// TIA Portal project "voda" (V17)

(* hardware
DEVICE "S71500/ET200MP-Station_1"  S7-1500 station
   slot 0: "Profilschiene_0"  6ES7 590-1***0-0AA0
   slot 1: "PLC_1"  CPU 1511-1 PN  6ES7 511-1AK00-0AB0  V1.8
   slot 2: "AI 8xU/I/RTD/TC ST_1"  AI 8xU/I/RTD/TC ST  6ES7 531-7KF00-0AB0  V2.0
   slot 3: "AI 8xU/I/RTD/TC ST_2"  AI 8xU/I/RTD/TC ST  6ES7 531-7KF00-0AB0  V2.0
   slot 4: "AI 8xU/I/RTD/TC ST_3"  AI 8xU/I/RTD/TC ST  6ES7 531-7KF00-0AB0  V2.0
   slot 5: "AI 8xU/I/RTD/TC ST_4"  AI 8xU/I/RTD/TC ST  6ES7 531-7KF00-0AB0  V2.0
   slot 6: "DI 16x24VDC BA_1"  DI 16x24VDC BA  6ES7 521-1BH10-0AA0  V1.0
DEVICE "HMI_1"  KTP700 Basic PN
   slot 0: "HMI_1"  KTP700 Basic PN  6AV2 123-2GB03-0AX0  17.0.0.0
   slot 1: "HMI_RT_1"  KTP700 Basic PN  6AV2 123-2GB03-0AX0  17.0.0.0
   slot 5: "HMI_1.IE_CP_1"  PROFINET Interface  17.0.0.0
      slot 1: "PROFINET Interface_1"  PROFINET Interface
         slot 1: "Port_1"  Port
*)

// ===== PLC "PLC_1"  CPU 1511-1 PN =====

VAR_GLOBAL   // PLC tag table "Standard-Variablentabelle"
   "Start" AT %I0.0 : Bool;
   "Reset" AT %I0.1 : Bool;
   "Stop" AT %I0.2 : Bool;
   "Factory_I/O" AT %I0.3 : Bool;
   "Level_Meter" AT %ID30 : Real;
   "Flow_Meter" AT %ID34 : Real;
   "Set_Point" AT %ID38 : Real;
   "Start_Light" AT %Q0.0 : Bool;
   "Reset_Light" AT %Q0.1 : Bool;
   "Stop_Light" AT %Q0.2 : Bool;
   "Fill_valve" AT %QD30 : Real;
   "Discharge_valve" AT %QD34 : Real;
   "SP" AT %QD38 : DInt;
   "PV" AT %QD42 : DInt;
   "Tag_1" AT %M0.0 : Bool;
   "Tag_2" AT %M100.2 : Bool;
   "Tag_3" AT %M600.0 : Bool;
   "Tag_4" AT %M20.0 : Bool;
   "Tag_5" AT %M20.1 : Bool;
   "Tag_6" AT %M20.2 : Bool;
END_VAR

DATA_BLOCK "global"   // DB1
{ S7_Optimized_Access := 'TRUE' }
VERSION : 0.1
   VAR
      POM : Array[0..100] of Bool;
      POM_BR : Array[0..100] of Real;
      SP_Real : Real;
      PV_Real : Real;
      Kp_Level : Real;
      Ki_Level : Real;
      Kp_Flow : Real;
      Ki_Flow : Real;
      Flow_Real : Real;
      Discharge_Real : Real;
      SP_flow : Real;
      "LevelSetPoint%" : Real;
      "FlowSP%" : Real;
      "FlowPV%" : Real;
      "LevelPV%" : Real;
      PV_flow : Real;
      FactoryIOPTrig : Bool;
      PID_CompactMode : Int := 3;
      "FlowSP0-10" : Real;
   END_VAR
BEGIN
END_DATA_BLOCK

DATA_BLOCK "PID_Level"   // DB2
{ S7_Optimized_Access := 'TRUE' }
VERSION : 0.1
// stored: InstanceOfName Block_3
"Block_3"
BEGIN
END_DATA_BLOCK

DATA_BLOCK "PID_Flow"   // DB3
{ S7_Optimized_Access := 'TRUE' }
VERSION : 0.1
// stored: InstanceOfName Block_3
"Block_3"
BEGIN
END_DATA_BLOCK

DATA_BLOCK "HMI Tags"   // DB7
{ S7_Optimized_Access := 'TRUE' }
VERSION : 0.1
   VAR
      PV_Level : Real;
      SP_Level : Real;
      "SP_Flow%" : DInt;
      PV_Flow : DInt;
      "SP_Level%" : Real;
      LevelSetPointInCM : Bool;
      "LevelSetPointIn%" : Bool;
      LevelSetpointInCMButton : Bool;
      "LevelSetpointIn%Button" : Bool;
      HMIButton : Bool;
      FactoryIOButton : Bool;
      HMI : Bool;
      FactoryIO : Bool;
      HMISPLevelSet : Real;
      "HMISPLevelSet%" : Real;
      "Dozvoljeno%" : Bool;
      DozvoljenoCM : Bool;
      Warning : Bool;
      LL_Alarm : Bool;
      L_Alarm : Bool;
      H_Alarm : Bool;
      HH_Alarm : Bool;
      LL_Pom : Bool;
      Level_0 : Bool;
      HH_Pom : Bool;
      ACKButton : Bool;
      ACK : Bool;
   END_VAR
BEGIN
END_DATA_BLOCK

FUNCTION_BLOCK "Block_3"   // FB1, SCL
{ S7_Optimized_Access := 'TRUE' }
VERSION : 0.1
   VAR_INPUT
      SP : Real;
      PV : Real;
      Kp : Real;
      Ki : Real;
      Xi_max : Real;
      "dt" : Real;
      Xi_min : Real;
   END_VAR
   VAR_OUTPUT
      U : Real;
   END_VAR
   VAR
      I : Real;
      Xi : Real;
      error : Real;
   END_VAR
BEGIN
   #I := 0;
   #error := #SP - #PV;
   #I := #I + #error * #dt;
   #Xi := (#Kp * #error) + (#Ki * #I);
   IF #Xi > #Xi_max THEN
       #U := #Xi_max;
       #I := #I - #error * #dt;
   ELSIF #Xi < #Xi_min THEN
       #U := #Xi_min;
       #I := #I - #error * #dt;
   ELSE
       #U := #Xi;
   END_IF;
END_FUNCTION_BLOCK

FUNCTION "Block_1" : Void   // FC1, LAD
{ S7_Optimized_Access := 'TRUE' }
VERSION : 0.1
   VAR_TEMP   // added for the SCL form of the ladder/FBD networks
      _w1 : Bool;
      _w2 : Bool;
   END_VAR
BEGIN

REGION Network 1
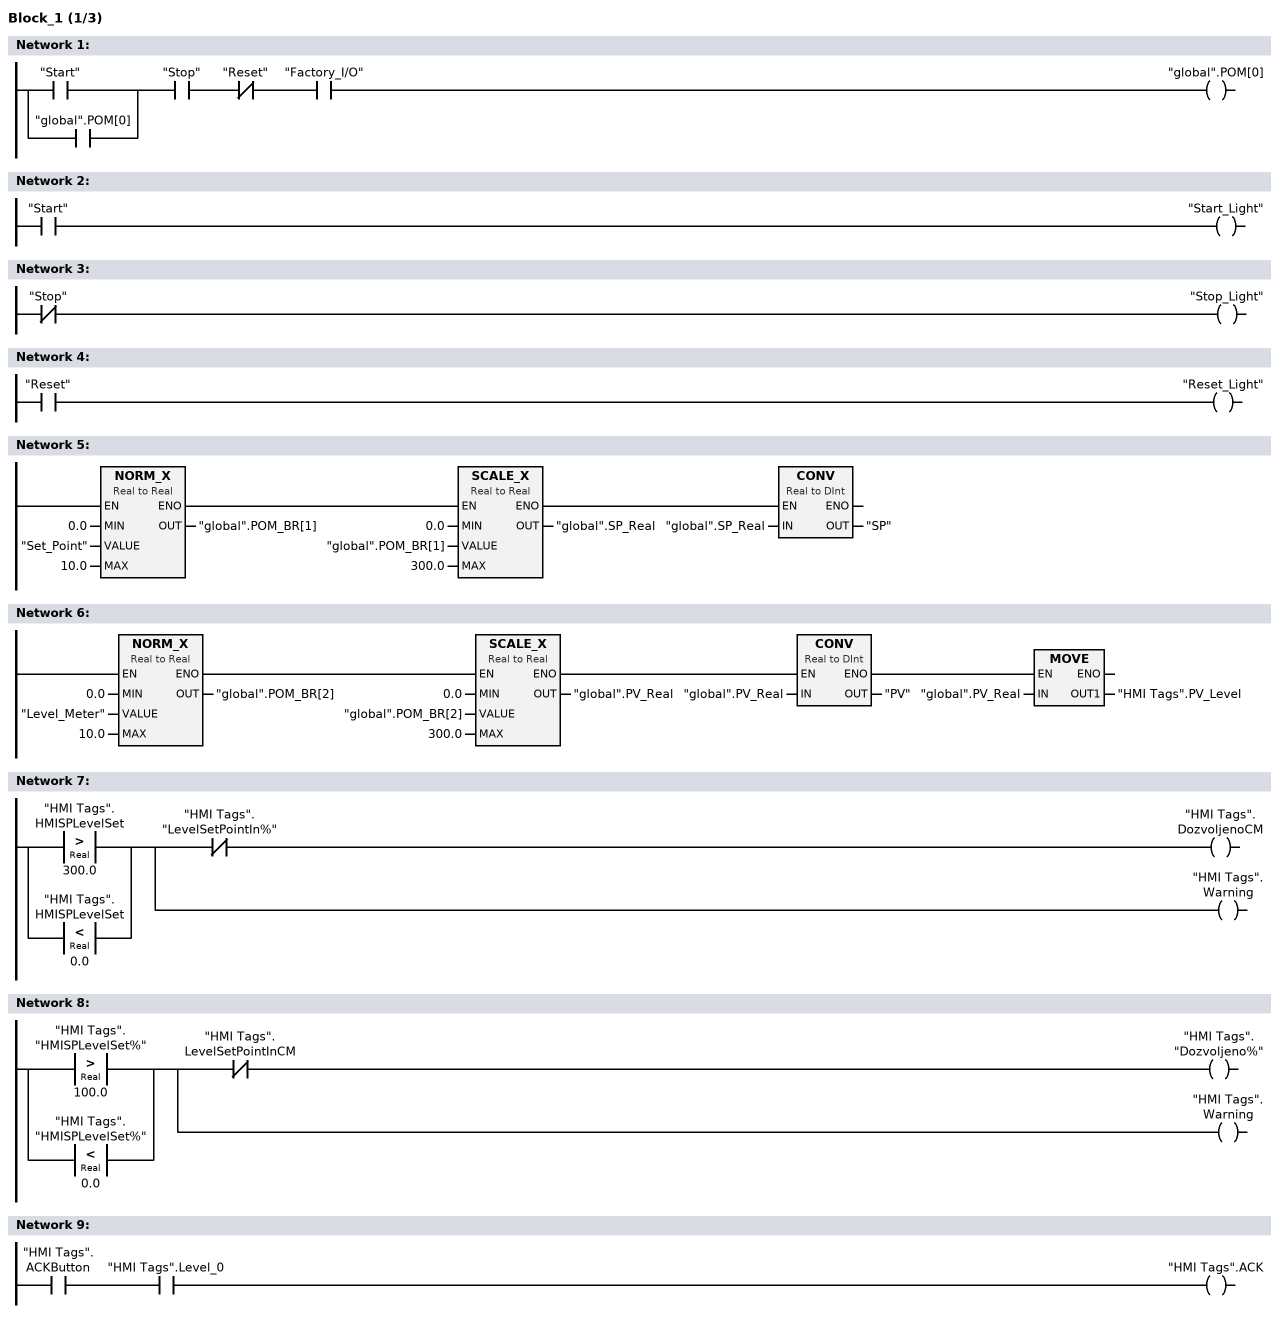
   RUNG wire#powerrail
      Contact( "Start" )
      wire#w1
      Contact( "Stop" )
      I_Contact( "Reset" )
      Contact( "Factory_I/O" )
      Coil( "global".POM[0] )
   END_RUNG
   RUNG wire#powerrail
      Contact( "global".POM[0] )
   END_RUNG wire#w1
   // the same network as SCL:
   "global".POM[0] := ("Start" OR "global".POM[0]) AND "Stop" AND NOT "Reset" AND "Factory_I/O";
END_REGION

REGION Network 2
   RUNG wire#powerrail
      Contact( "Start" )
      Coil( "Start_Light" )
   END_RUNG
   // the same network as SCL:
   "Start_Light" := "Start";
END_REGION

REGION Network 3
   RUNG wire#powerrail
      I_Contact( "Stop" )
      Coil( "Stop_Light" )
   END_RUNG
   // the same network as SCL:
   "Stop_Light" := NOT "Stop";
END_REGION

REGION Network 4
   RUNG wire#powerrail
      Contact( "Reset" )
      Coil( "Reset_Light" )
   END_RUNG
   // the same network as SCL:
   "Reset_Light" := "Reset";
END_REGION

REGION Network 5
   RUNG wire#powerrail
      { S7_Templates := "[SrcType := Real, DestType := Real]" } Normalize(min := 0.0, value := "Set_Point", max := 10.0, out => "global".POM_BR[1])
      { S7_Templates := "[SrcType := Real, DestType := Real]" } Scale(min := 0.0, value := "global".POM_BR[1], max := 300.0, out => "global".SP_Real)
      { S7_Templates := "[SrcType := Real, DestType := DInt]" } Convert(in := "global".SP_Real, out => "SP")
   END_RUNG
   // the same network as SCL:
   "global".POM_BR[1] := NORM_X(MIN := 0.0, VALUE := "Set_Point", MAX := 10.0);
   "global".SP_Real := SCALE_X(MIN := 0.0, VALUE := "global".POM_BR[1], MAX := 300.0);
   "SP" := REAL_TO_DINT("global".SP_Real);
END_REGION

REGION Network 6
   RUNG wire#powerrail
      { S7_Templates := "[SrcType := Real, DestType := Real]" } Normalize(min := 0.0, value := "Level_Meter", max := 10.0, out => "global".POM_BR[2])
      { S7_Templates := "[SrcType := Real, DestType := Real]" } Scale(min := 0.0, value := "global".POM_BR[2], max := 300.0, out => "global".PV_Real)
      { S7_Templates := "[SrcType := Real, DestType := DInt]" } Convert(in := "global".PV_Real, out => "PV")
      Move(in := "global".PV_Real, out1 => "HMI Tags".PV_Level)
   END_RUNG
   // the same network as SCL:
   "global".POM_BR[2] := NORM_X(MIN := 0.0, VALUE := "Level_Meter", MAX := 10.0);
   "global".PV_Real := SCALE_X(MIN := 0.0, VALUE := "global".POM_BR[2], MAX := 300.0);
   "PV" := REAL_TO_DINT("global".PV_Real);
   "HMI Tags".PV_Level := "global".PV_Real;
END_REGION

REGION Network 7
   RUNG wire#powerrail
      { S7_Templates := "SrcType := Real" } GT_Contact(in1 := "HMI Tags".HMISPLevelSet, in2 := 300.0)
      wire#w1
      I_Contact( "HMI Tags"."LevelSetPointIn%" )
      Coil( "HMI Tags".DozvoljenoCM )
   END_RUNG
   RUNG wire#powerrail
      { S7_Templates := "SrcType := Real" } LT_Contact(in1 := "HMI Tags".HMISPLevelSet, in2 := 0.0)
   END_RUNG wire#w1
   RUNG wire#w1
      Coil( "HMI Tags".Warning )
   END_RUNG
   // the same network as SCL:
   #_w1 := ("HMI Tags".HMISPLevelSet > 300.0) OR ("HMI Tags".HMISPLevelSet < 0.0);
   "HMI Tags".DozvoljenoCM := #_w1 AND NOT "HMI Tags"."LevelSetPointIn%";
   "HMI Tags".Warning := #_w1;
END_REGION

REGION Network 8
   RUNG wire#powerrail
      { S7_Templates := "SrcType := Real" } GT_Contact(in1 := "HMI Tags"."HMISPLevelSet%", in2 := 100.0)
      wire#w1
      I_Contact( "HMI Tags".LevelSetPointInCM )
      Coil( "HMI Tags"."Dozvoljeno%" )
   END_RUNG
   RUNG wire#powerrail
      { S7_Templates := "SrcType := Real" } LT_Contact(in1 := "HMI Tags"."HMISPLevelSet%", in2 := 0.0)
   END_RUNG wire#w1
   RUNG wire#w1
      Coil( "HMI Tags".Warning )
   END_RUNG
   // the same network as SCL:
   #_w1 := ("HMI Tags"."HMISPLevelSet%" > 100.0) OR ("HMI Tags"."HMISPLevelSet%" < 0.0);
   "HMI Tags"."Dozvoljeno%" := #_w1 AND NOT "HMI Tags".LevelSetPointInCM;
   "HMI Tags".Warning := #_w1;
END_REGION

REGION Network 9
   RUNG wire#powerrail
      Contact( "HMI Tags".ACKButton )
      Contact( "HMI Tags".Level_0 )
      Coil( "HMI Tags".ACK )
   END_RUNG
   // the same network as SCL:
   "HMI Tags".ACK := "HMI Tags".ACKButton AND "HMI Tags".Level_0;
END_REGION

REGION Network 10
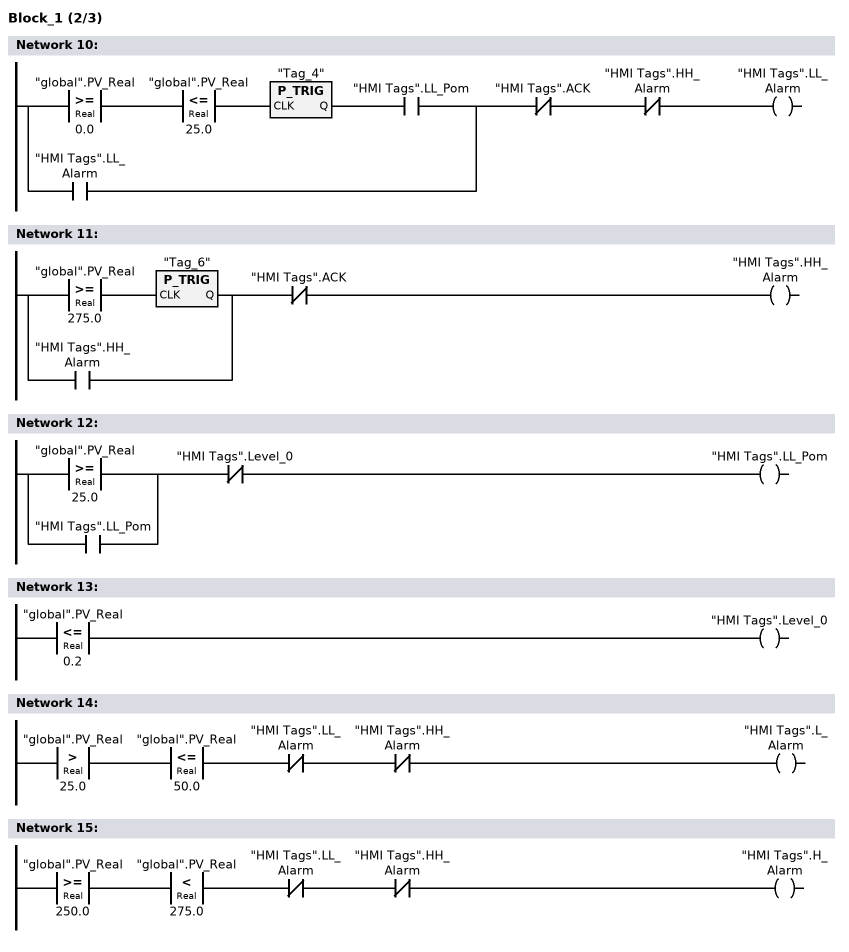
   RUNG wire#powerrail
      { S7_Templates := "SrcType := Real" } GE_Contact(in1 := "global".PV_Real, in2 := 0.0)
      { S7_Templates := "SrcType := Real" } LE_Contact(in1 := "global".PV_Real, in2 := 25.0)
      P_Trig( "Tag_4" )
      Contact( "HMI Tags".LL_Pom )
      wire#w1
      I_Contact( "HMI Tags".ACK )
      I_Contact( "HMI Tags".HH_Alarm )
      Coil( "HMI Tags".LL_Alarm )
   END_RUNG
   RUNG wire#powerrail
      Contact( "HMI Tags".LL_Alarm )
   END_RUNG wire#w1
   // the same network as SCL:
   #_w1 := ("global".PV_Real >= 0.0) AND ("global".PV_Real <= 25.0);
   #_w2 := #_w1 AND NOT "Tag_4";   // rising edge
   "Tag_4" := #_w1;
   "HMI Tags".LL_Alarm := ((#_w2 AND "HMI Tags".LL_Pom) OR "HMI Tags".LL_Alarm) AND NOT "HMI Tags".ACK AND NOT "HMI Tags".HH_Alarm;
END_REGION

REGION Network 11
   RUNG wire#powerrail
      { S7_Templates := "SrcType := Real" } GE_Contact(in1 := "global".PV_Real, in2 := 275.0)
      P_Trig( "Tag_6" )
      wire#w1
      I_Contact( "HMI Tags".ACK )
      Coil( "HMI Tags".HH_Alarm )
   END_RUNG
   RUNG wire#powerrail
      Contact( "HMI Tags".HH_Alarm )
   END_RUNG wire#w1
   // the same network as SCL:
   #_w1 := "global".PV_Real >= 275.0;
   #_w2 := #_w1 AND NOT "Tag_6";   // rising edge
   "Tag_6" := #_w1;
   "HMI Tags".HH_Alarm := (#_w2 OR "HMI Tags".HH_Alarm) AND NOT "HMI Tags".ACK;
END_REGION

REGION Network 12
   RUNG wire#powerrail
      { S7_Templates := "SrcType := Real" } GE_Contact(in1 := "global".PV_Real, in2 := 25.0)
      wire#w1
      I_Contact( "HMI Tags".Level_0 )
      Coil( "HMI Tags".LL_Pom )
   END_RUNG
   RUNG wire#powerrail
      Contact( "HMI Tags".LL_Pom )
   END_RUNG wire#w1
   // the same network as SCL:
   "HMI Tags".LL_Pom := (("global".PV_Real >= 25.0) OR "HMI Tags".LL_Pom) AND NOT "HMI Tags".Level_0;
END_REGION

REGION Network 13
   RUNG wire#powerrail
      { S7_Templates := "SrcType := Real" } LE_Contact(in1 := "global".PV_Real, in2 := 0.2)
      Coil( "HMI Tags".Level_0 )
   END_RUNG
   // the same network as SCL:
   "HMI Tags".Level_0 := "global".PV_Real <= 0.2;
END_REGION

REGION Network 14
   RUNG wire#powerrail
      { S7_Templates := "SrcType := Real" } GT_Contact(in1 := "global".PV_Real, in2 := 25.0)
      { S7_Templates := "SrcType := Real" } LE_Contact(in1 := "global".PV_Real, in2 := 50.0)
      I_Contact( "HMI Tags".LL_Alarm )
      I_Contact( "HMI Tags".HH_Alarm )
      Coil( "HMI Tags".L_Alarm )
   END_RUNG
   // the same network as SCL:
   "HMI Tags".L_Alarm := ("global".PV_Real > 25.0) AND ("global".PV_Real <= 50.0) AND NOT "HMI Tags".LL_Alarm AND NOT "HMI Tags".HH_Alarm;
END_REGION

REGION Network 15
   RUNG wire#powerrail
      { S7_Templates := "SrcType := Real" } GE_Contact(in1 := "global".PV_Real, in2 := 250.0)
      { S7_Templates := "SrcType := Real" } LT_Contact(in1 := "global".PV_Real, in2 := 275.0)
      I_Contact( "HMI Tags".LL_Alarm )
      I_Contact( "HMI Tags".HH_Alarm )
      Coil( "HMI Tags".H_Alarm )
   END_RUNG
   // the same network as SCL:
   "HMI Tags".H_Alarm := ("global".PV_Real >= 250.0) AND ("global".PV_Real < 275.0) AND NOT "HMI Tags".LL_Alarm AND NOT "HMI Tags".HH_Alarm;
END_REGION

REGION Network 16
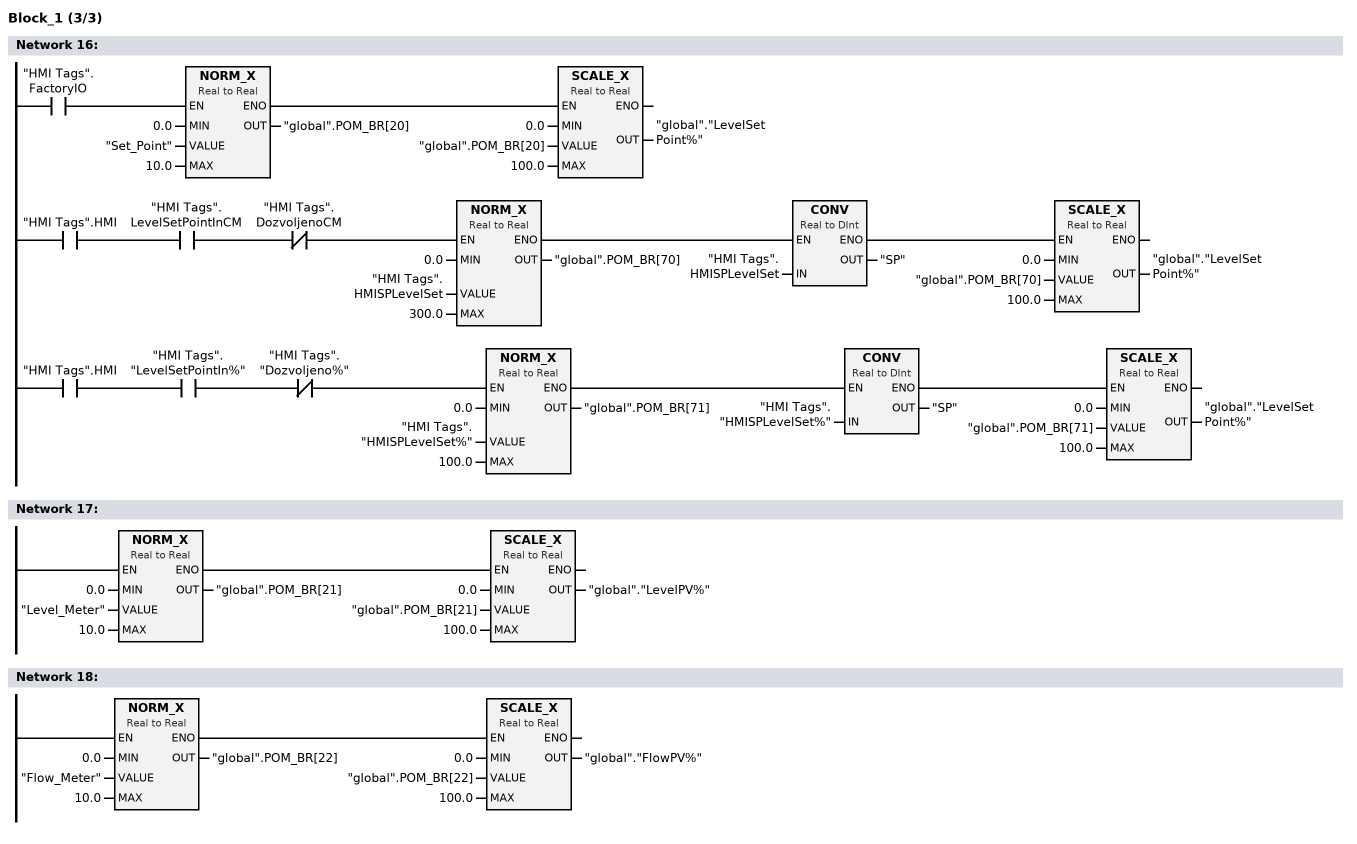
   RUNG wire#powerrail
      Contact( "HMI Tags".FactoryIO )
      { S7_Templates := "[SrcType := Real, DestType := Real]" } Normalize(min := 0.0, value := "Set_Point", max := 10.0, out => "global".POM_BR[20])
      { S7_Templates := "[SrcType := Real, DestType := Real]" } Scale(min := 0.0, value := "global".POM_BR[20], max := 100.0, out => "global"."LevelSetPoint%")
   END_RUNG
   RUNG wire#powerrail
      Contact( "HMI Tags".HMI )
      Contact( "HMI Tags".LevelSetPointInCM )
      I_Contact( "HMI Tags".DozvoljenoCM )
      { S7_Templates := "[SrcType := Real, DestType := Real]" } Normalize(min := 0.0, value := "HMI Tags".HMISPLevelSet, max := 300.0, out => "global".POM_BR[70])
      { S7_Templates := "[SrcType := Real, DestType := DInt]" } Convert(in := "HMI Tags".HMISPLevelSet, out => "SP")
      { S7_Templates := "[SrcType := Real, DestType := Real]" } Scale(min := 0.0, value := "global".POM_BR[70], max := 100.0, out => "global"."LevelSetPoint%")
   END_RUNG
   RUNG wire#powerrail
      Contact( "HMI Tags".HMI )
      Contact( "HMI Tags"."LevelSetPointIn%" )
      I_Contact( "HMI Tags"."Dozvoljeno%" )
      { S7_Templates := "[SrcType := Real, DestType := Real]" } Normalize(min := 0.0, value := "HMI Tags"."HMISPLevelSet%", max := 100.0, out => "global".POM_BR[71])
      { S7_Templates := "[SrcType := Real, DestType := DInt]" } Convert(in := "HMI Tags"."HMISPLevelSet%", out => "SP")
      { S7_Templates := "[SrcType := Real, DestType := Real]" } Scale(min := 0.0, value := "global".POM_BR[71], max := 100.0, out => "global"."LevelSetPoint%")
   END_RUNG
   // the same network as SCL:
   IF "HMI Tags".FactoryIO THEN
       "global".POM_BR[20] := NORM_X(MIN := 0.0, VALUE := "Set_Point", MAX := 10.0);
       "global"."LevelSetPoint%" := SCALE_X(MIN := 0.0, VALUE := "global".POM_BR[20], MAX := 100.0);
   END_IF;
   IF "HMI Tags".HMI AND "HMI Tags".LevelSetPointInCM AND NOT "HMI Tags".DozvoljenoCM THEN
       "global".POM_BR[70] := NORM_X(MIN := 0.0, VALUE := "HMI Tags".HMISPLevelSet, MAX := 300.0);
       "SP" := REAL_TO_DINT("HMI Tags".HMISPLevelSet);
       "global"."LevelSetPoint%" := SCALE_X(MIN := 0.0, VALUE := "global".POM_BR[70], MAX := 100.0);
   END_IF;
   IF "HMI Tags".HMI AND "HMI Tags"."LevelSetPointIn%" AND NOT "HMI Tags"."Dozvoljeno%" THEN
       "global".POM_BR[71] := NORM_X(MIN := 0.0, VALUE := "HMI Tags"."HMISPLevelSet%", MAX := 100.0);
       "SP" := REAL_TO_DINT("HMI Tags"."HMISPLevelSet%");
       "global"."LevelSetPoint%" := SCALE_X(MIN := 0.0, VALUE := "global".POM_BR[71], MAX := 100.0);
   END_IF;
END_REGION

REGION Network 17
   RUNG wire#powerrail
      { S7_Templates := "[SrcType := Real, DestType := Real]" } Normalize(min := 0.0, value := "Level_Meter", max := 10.0, out => "global".POM_BR[21])
      { S7_Templates := "[SrcType := Real, DestType := Real]" } Scale(min := 0.0, value := "global".POM_BR[21], max := 100.0, out => "global"."LevelPV%")
   END_RUNG
   // the same network as SCL:
   "global".POM_BR[21] := NORM_X(MIN := 0.0, VALUE := "Level_Meter", MAX := 10.0);
   "global"."LevelPV%" := SCALE_X(MIN := 0.0, VALUE := "global".POM_BR[21], MAX := 100.0);
END_REGION

REGION Network 18
   RUNG wire#powerrail
      { S7_Templates := "[SrcType := Real, DestType := Real]" } Normalize(min := 0.0, value := "Flow_Meter", max := 10.0, out => "global".POM_BR[22])
      { S7_Templates := "[SrcType := Real, DestType := Real]" } Scale(min := 0.0, value := "global".POM_BR[22], max := 100.0, out => "global"."FlowPV%")
   END_RUNG
   // the same network as SCL:
   "global".POM_BR[22] := NORM_X(MIN := 0.0, VALUE := "Flow_Meter", MAX := 10.0);
   "global"."FlowPV%" := SCALE_X(MIN := 0.0, VALUE := "global".POM_BR[22], MAX := 100.0);
END_REGION
END_FUNCTION

FUNCTION "HMI" : Void   // FC2, LAD
{ S7_Optimized_Access := 'TRUE' }
VERSION : 0.1
BEGIN

REGION Network 1
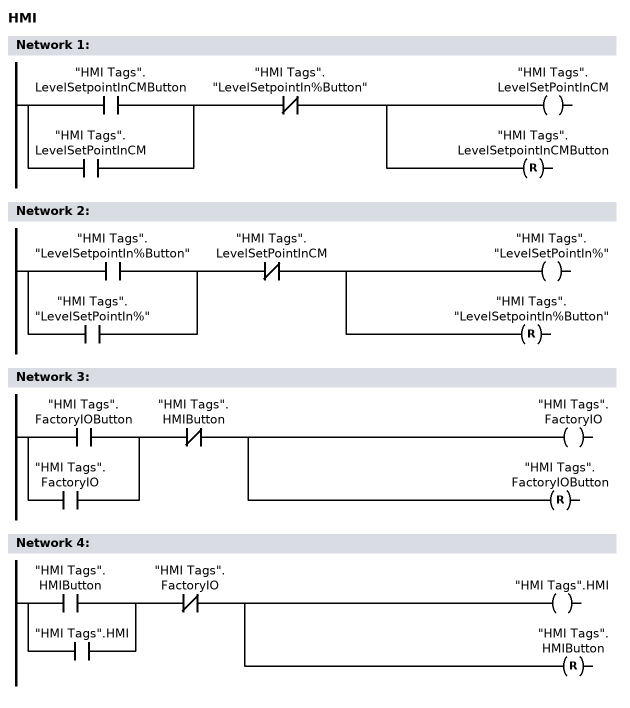
   RUNG wire#powerrail
      Contact( "HMI Tags".LevelSetpointInCMButton )
      wire#w1
      I_Contact( "HMI Tags"."LevelSetpointIn%Button" )
      wire#w2
      Coil( "HMI Tags".LevelSetPointInCM )
   END_RUNG
   RUNG wire#powerrail
      Contact( "HMI Tags".LevelSetPointInCM )
   END_RUNG wire#w1
   RUNG wire#w2
      R_Coil( "HMI Tags".LevelSetpointInCMButton )
   END_RUNG
   // the same network as SCL:
   "HMI Tags".LevelSetPointInCM := ("HMI Tags".LevelSetpointInCMButton OR "HMI Tags".LevelSetPointInCM) AND NOT "HMI Tags"."LevelSetpointIn%Button";
   IF "HMI Tags".LevelSetPointInCM THEN "HMI Tags".LevelSetpointInCMButton := FALSE; END_IF;
END_REGION

REGION Network 2
   RUNG wire#powerrail
      Contact( "HMI Tags"."LevelSetpointIn%Button" )
      wire#w1
      I_Contact( "HMI Tags".LevelSetPointInCM )
      wire#w2
      Coil( "HMI Tags"."LevelSetPointIn%" )
   END_RUNG
   RUNG wire#powerrail
      Contact( "HMI Tags"."LevelSetPointIn%" )
   END_RUNG wire#w1
   RUNG wire#w2
      R_Coil( "HMI Tags"."LevelSetpointIn%Button" )
   END_RUNG
   // the same network as SCL:
   "HMI Tags"."LevelSetPointIn%" := ("HMI Tags"."LevelSetpointIn%Button" OR "HMI Tags"."LevelSetPointIn%") AND NOT "HMI Tags".LevelSetPointInCM;
   IF "HMI Tags"."LevelSetPointIn%" THEN "HMI Tags"."LevelSetpointIn%Button" := FALSE; END_IF;
END_REGION

REGION Network 3
   RUNG wire#powerrail
      Contact( "HMI Tags".FactoryIOButton )
      wire#w1
      I_Contact( "HMI Tags".HMIButton )
      wire#w2
      Coil( "HMI Tags".FactoryIO )
   END_RUNG
   RUNG wire#powerrail
      Contact( "HMI Tags".FactoryIO )
   END_RUNG wire#w1
   RUNG wire#w2
      R_Coil( "HMI Tags".FactoryIOButton )
   END_RUNG
   // the same network as SCL:
   "HMI Tags".FactoryIO := ("HMI Tags".FactoryIOButton OR "HMI Tags".FactoryIO) AND NOT "HMI Tags".HMIButton;
   IF "HMI Tags".FactoryIO THEN "HMI Tags".FactoryIOButton := FALSE; END_IF;
END_REGION

REGION Network 4
   RUNG wire#powerrail
      Contact( "HMI Tags".HMIButton )
      wire#w1
      I_Contact( "HMI Tags".FactoryIO )
      wire#w2
      Coil( "HMI Tags".HMI )
   END_RUNG
   RUNG wire#powerrail
      Contact( "HMI Tags".HMI )
   END_RUNG wire#w1
   RUNG wire#w2
      R_Coil( "HMI Tags".HMIButton )
   END_RUNG
   // the same network as SCL:
   "HMI Tags".HMI := ("HMI Tags".HMIButton OR "HMI Tags".HMI) AND NOT "HMI Tags".FactoryIO;
   IF "HMI Tags".HMI THEN "HMI Tags".HMIButton := FALSE; END_IF;
END_REGION
END_FUNCTION

FUNCTION "MHJ-PLC-Lab-Function-S71500" : Void   // FC9000, SCL
{ S7_Optimized_Access := 'TRUE' }
VERSION : 0.1
   VAR_TEMP
      Value : Byte;
      ForCounter : Int;
   END_VAR
   VAR CONSTANT
      Value_01_DW : DWord := 16#1223_5486;
      Value_02_DW : DWord := 16#A6C9_D1F5;
   END_VAR
BEGIN

   #Value:=PEEK(area := 16#82,
        dbNumber := 0,
        byteOffset := 511);
   #Value := #Value + 1;

   POKE(area := 16#82,
        dbNumber := 0,
        byteOffset := 511,
        value := #Value);

   POKE(area := 16#82,
        dbNumber := 0,
        byteOffset := 1016,
        value := #Value_01_DW);
   POKE(area := 16#82,
        dbNumber := 0,
        byteOffset := 1020,
        value := #Value_02_DW);

   FOR #ForCounter := 0 TO 63 DO
       #Value:=PEEK(area := 16#1,
            dbNumber := 0,
            byteOffset := #ForCounter);
       POKE(area := 16#81,
            dbNumber := 0,
            byteOffset := #ForCounter,
            value := #Value);
   END_FOR;
   #Value := PEEK(area := 16#1,
                  dbNumber := 0,
                  byteOffset := 512);
   POKE(area := 16#82,
        dbNumber := 0,
        byteOffset := 512,
        value := #Value);
END_FUNCTION

ORGANIZATION_BLOCK "Main"   // OB1, FBD, ProgramCycle
TITLE = "Main Program Sweep (Cycle)"
{ S7_Optimized_Access := 'TRUE' }
VERSION : 0.1
   VAR_INPUT
      Initial_Call : Bool;   // Initial call of this OB
      Remanence : Bool;   // =True, if remanent data are available
   END_VAR
BEGIN

REGION Network 1
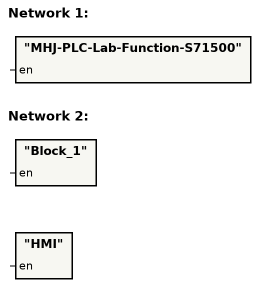
   "MHJ-PLC-Lab-Function-S71500"();
END_REGION

REGION Network 2
   "Block_1"();
   "HMI"();
END_REGION
END_ORGANIZATION_BLOCK

ORGANIZATION_BLOCK "PI kontroler"   // OB30, LAD, CyclicInterrupt
{ S7_Optimized_Access := 'TRUE' }
VERSION : 0.1
   VAR_INPUT
      Initial_Call : Bool;   // Initial call of this OB
      Event_Count : Int;   // Events discarded
   END_VAR
   VAR_TEMP   // added for the SCL form of the ladder/FBD networks
      _w1 : Bool;
   END_VAR
BEGIN

REGION Network 1
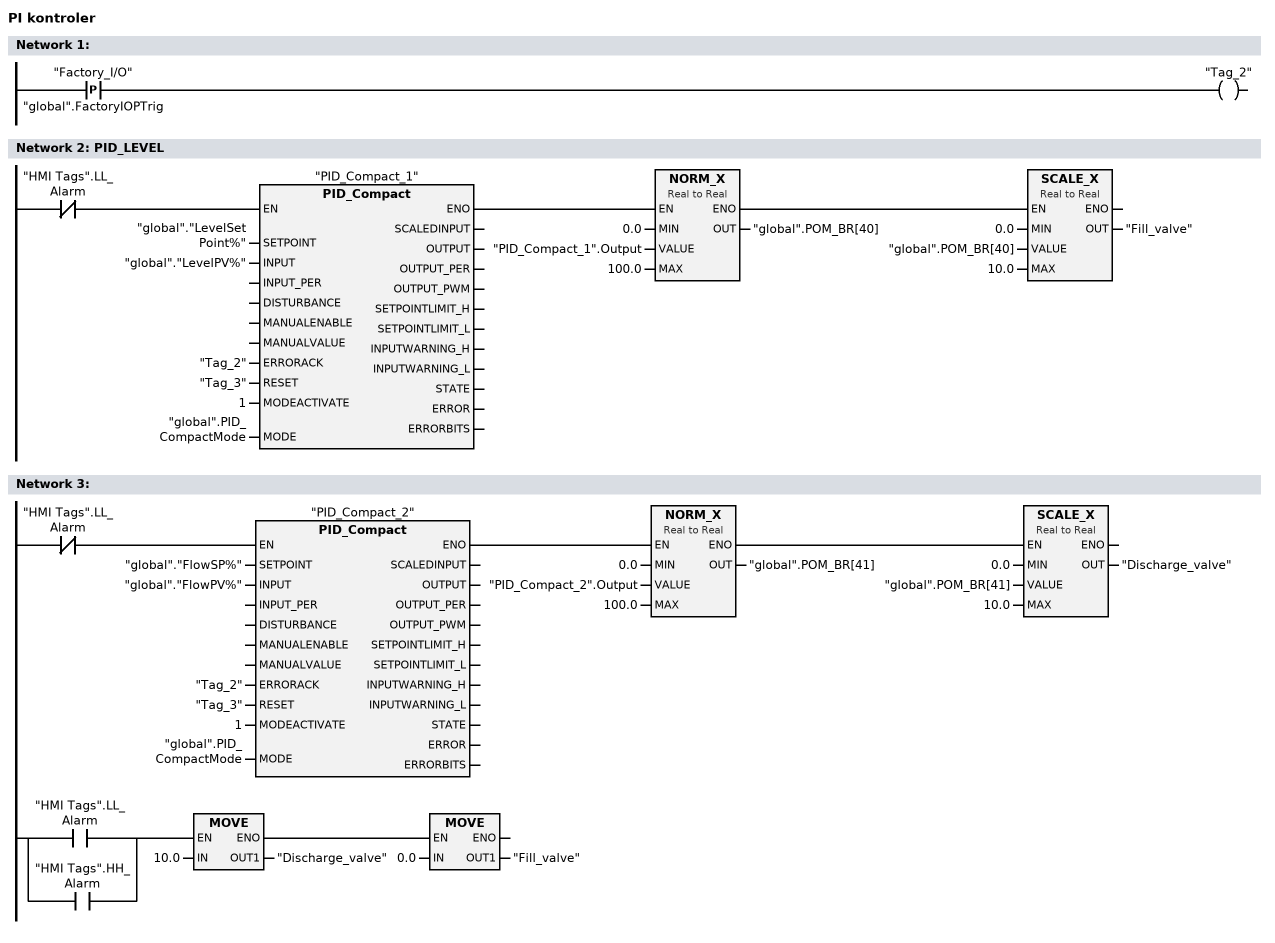
   RUNG wire#powerrail
      P_Contact(operand := "Factory_I/O", bit := "global".FactoryIOPTrig)
      Coil( "Tag_2" )
   END_RUNG
   // the same network as SCL:
   #_w1 := "Factory_I/O" AND NOT "global".FactoryIOPTrig;   // rising edge of "Factory_I/O"
   "global".FactoryIOPTrig := "Factory_I/O";
   "Tag_2" := #_w1;
END_REGION

REGION Network 2: PID_LEVEL
   // ENO of a box is taken as its EN; it also drops when the box reports an error
   #_w1 := NOT "HMI Tags".LL_Alarm;
   IF #_w1 THEN
       "PID_Compact_1"(Setpoint := "global"."LevelSetPoint%",   // PID_Compact
                       Input := "global"."LevelPV%",
                       ErrorAck := "Tag_2",
                       Reset := "Tag_3",
                       ModeActivate := 1,
                       Mode := "global".PID_CompactMode);
       "global".POM_BR[40] := NORM_X(MIN := 0.0, VALUE := "PID_Compact_1".Output, MAX := 100.0);
       "Fill_valve" := SCALE_X(MIN := 0.0, VALUE := "global".POM_BR[40], MAX := 10.0);
   END_IF;
END_REGION

REGION Network 3
   // ENO of a box is taken as its EN; it also drops when the box reports an error
   #_w1 := NOT "HMI Tags".LL_Alarm;
   IF #_w1 THEN
       "PID_Compact_2"(Setpoint := "global"."FlowSP%",   // PID_Compact
                       Input := "global"."FlowPV%",
                       ErrorAck := "Tag_2",
                       Reset := "Tag_3",
                       ModeActivate := 1,
                       Mode := "global".PID_CompactMode);
       "global".POM_BR[41] := NORM_X(MIN := 0.0, VALUE := "PID_Compact_2".Output, MAX := 100.0);
       "Discharge_valve" := SCALE_X(MIN := 0.0, VALUE := "global".POM_BR[41], MAX := 10.0);
   END_IF;
   IF "HMI Tags".LL_Alarm OR "HMI Tags".HH_Alarm THEN
       "Discharge_valve" := 10.0;
       "Fill_valve" := 0.0;
   END_IF;
END_REGION
END_ORGANIZATION_BLOCK

(* ===== HMI "HMI_RT_1" =====
system functions are stored by id; their names below are inferred from use
connection "Connection_1": ETHERNET, SMART_S7_1200_OMS
connection "HMI_Connection_1": ETHERNET, SMART_S7_1500_OMS

HMI tags "Default tag table"
   "HMI Tags_PV_Level" : Real = PLC "HMI Tags".PV_Level, 1 s
   "HMI Tags_SP_Level" : Real = PLC "HMI Tags".SP_Level, 1 s
   "HMI Tags_SP_Level%" : Real = PLC "HMI Tags".SP_Level%, 1 s
   "HMI Tags_LevelSetpointInCMButton" : Bool = PLC "HMI Tags".LevelSetpointInCMButton, 1 s
   "HMI Tags_HMI/FIO" : Bool = PLC "HMI Tags".HMIButton, 1 s
   "HMI Tags_FactoryIOButton" : Bool = PLC "HMI Tags".FactoryIOButton, 1 s
   "HMI Tags_HMISPLevelSet" : Real = PLC "HMI Tags".HMISPLevelSet, 1 s
   "HMI Tags_LevelSetpointIn%Button" : Bool = PLC "HMI Tags".LevelSetpointIn%Button, 1 s
   "HMI Tags_LevelSetPointInCM" : Bool = PLC "HMI Tags".LevelSetPointInCM, 1 s
   "HMI Tags_LevelSetPointIn%" : Bool = PLC "HMI Tags".LevelSetPointIn%, 1 s
   "HMI Tags_HMISPLevelSet%" : Real = PLC "HMI Tags".HMISPLevelSet%, 1 s
   "HMI Tags_Dozvoljeno%" : Bool = PLC "HMI Tags".Dozvoljeno%, 1 s
   "HMI Tags_DozvoljenoCM" : Bool = PLC "HMI Tags".DozvoljenoCM, 1 s
   "HMI Tags_FactoryIO" : Bool = PLC "HMI Tags".FactoryIO, 1 s
   "HMI Tags_HMI" : Bool = PLC "HMI Tags".HMI, 1 s
   "global_FlowSP%" : Real = PLC global.FlowSP%, 1 s
   "HMI Tags_Warning" : Bool = PLC "HMI Tags".Warning, 1 s
   "HMI Tags_LL_Alarm" : Bool = PLC "HMI Tags".LL_Alarm, 1 s
   "HMI Tags_L_Alarm" : Bool = PLC "HMI Tags".L_Alarm, 1 s
   "HMI Tags_H_Alarm" : Bool = PLC "HMI Tags".H_Alarm, 1 s
   "HMI Tags_HH_Alarm" : Bool = PLC "HMI Tags".HH_Alarm, 1 s
   "HMI Tags_ACK" : Bool = PLC "HMI Tags".ACK, 1 s
   "HMI Tags_ACKButton" : Bool = PLC "HMI Tags".ACKButton, 1 s
   "global_FlowPV%" : Real = PLC global.FlowPV%, 1 s
   "HMI Tags_LL_Pom" : Bool = PLC "HMI Tags".LL_Pom, 1 s

screen "Screen_1" 800x480
   GraphicView "Graphic view_1" at 44,86 size 267x322; Picture "Graphic_2"
   Bar "Bar_1" at 55,108 size 239x284; MinimumValue 0; MaximumValue 300
      ProcessValue <- "HMI Tags_PV_Level"
   IOField "I/O field_1" at 446,165 size 54x38; FormatPattern 999
      ProcessValue <- "HMI Tags_HMISPLevelSet"
      Visibility <- "HMI Tags_LevelSetPointInCM"
   TextField "Text field_1" at 431,134 size 102x20; Text 'Set Point in CM'
      Visibility <- "HMI Tags_LevelSetPointInCM"
   IOField "I/O field_2" at 337,165 size 66x39; FormatPattern 999
      ProcessValue <- "HMI Tags_PV_Level"
   TextField "Text field_2" at 328,134 size 95x20; Text 'Process value'
   Button "Button_1" at 364,365 size 136x62; TextOff 'HMI'
      on Click: SetBit("HMI Tags_HMI/FIO")
      Appearance <- "HMI Tags_HMI"
   Button "Button_2" at 364,270 size 136x62; TextOff 'Factory'
      on Click: SetBit("HMI Tags_FactoryIOButton")
      Appearance <- "HMI Tags_FactoryIO"
   Button "Button_3" at 611,365 size 136x62; TextOff 'IN CM'
      on Click: SetBit("HMI Tags_LevelSetpointInCMButton")
      Appearance <- "HMI Tags_LevelSetPointInCM"
   Button "Button_4" at 610,271 size 136x62; TextOff 'IN %'
      on Click: SetBit("HMI Tags_LevelSetpointIn%Button")
      Appearance <- "HMI Tags_LevelSetPointIn%"
   IOField "I/O field_3" at 446,165 size 60x38; FormatPattern 999
      ProcessValue <- "HMI Tags_HMISPLevelSet%"
      Visibility <- "HMI Tags_LevelSetPointIn%"
   TextField "Text field_3" at 431,134 size 97x20; Text 'Set Point in %'
      Visibility <- "HMI Tags_LevelSetPointIn%"
   IOField "I/O field_4" at 550,166 size 49x38; FormatPattern 999
      ProcessValue <- "global_FlowSP%"
   TextField "Text field_6" at 550,134 size 86x20; Text 'Flow SP in %'
   TextField "Text field_4" at 151,42 size 448x37; Text 'CHOOSE VALUE BETWEEN 0-100'
      Visibility <- "HMI Tags_Dozvoljeno%"
   TextField "Text field_5" at 151,42 size 448x37; Text 'CHOOSE VALUE BETWEEN 0-300'
      Visibility <- "HMI Tags_DozvoljenoCM"
   Rectangle "Rectangle_1" at 151,2 size 456x73
      Visibility <- "HMI Tags_Warning"
   TextField "Text field_8" at 488,99 size 143x29; Text 'Value control'
   TextField "Text field_9" at 583,235 size 191x27; Text 'Value mode control'
   TextField "Text field_10" at 329,235 size 202x27; Text 'Factory/HMI control'
   Rectangle "Rectangle_5" at 8,359 size 37x35
      Appearance <- "HMI Tags_LL_Alarm"
   Rectangle "Rectangle_7" at 7,142 size 37x35
      Appearance <- "HMI Tags_H_Alarm"
   Rectangle "Rectangle_8" at 8,99 size 37x35
      Appearance <- "HMI Tags_HH_Alarm"
   TextField "Text field_11" at 12,105 size 29x23; Text 'HH'
   TextField "Text field_12" at 17,145 size 17x23; Text 'H'
   TextField "Text field_14" at 12,365 size 23x23; Text 'LL'
   Rectangle "Rectangle_6" at 7,314 size 37x35
      Appearance <- "HMI Tags_L_Alarm"
   TextField "Text field_13" at 20,320 size 14x23; Text 'L'
   Button "Button_5" at 112,419 size 103x37; TextOff 'ACK'
      on Press: SetBit("HMI Tags_ACKButton")
      on Release: ResetBit("HMI Tags_ACKButton")
   IOField "I/O field_5" at 671,165 size 66x38; FormatPattern 999
      ProcessValue <- "global_FlowPV%"
   TextField "Text field_15" at 666,134 size 54x20; Text 'Flow PV'
   TextField "Text field_16" at 167,8 size 416x37; Text 'Upper limit reached, emptying'
      Visibility <- "HMI Tags_HH_Alarm"
   TextField "Text field_17" at 168,8 size 418x37; Text 'Lower limit reached, emptying'
      Visibility <- "HMI Tags_LL_Alarm"
   TextField "Text field_18" at 248,8 size 249x37; Text 'Low level reached'
      Visibility <- "HMI Tags_L_Alarm"
   TextField "Text field_19" at 244,5 size 256x37; Text 'High level reached'
      Visibility <- "HMI Tags_H_Alarm"
*)